PROGRAM Pneumatics_Template_Shutter
VAR
    bExtendedLight AT %Q*: BOOL; //Power output for Open position + LED
    bRetractedLight AT %Q*: BOOL; //Power output for Close position + LED
    bMovingLight AT %Q*: BOOL; //Power output for cylinder Moving LED
    bNoPermitLight AT %Q*: BOOL; //Power output for No permit LED
    bErrorLight AT %Q*: BOOL; //Power output for Error LED
END_VAR

//Assign LED to the permit status
bNoPermitLight := NOT gvl.astPneumaticAxes[main.hmiPneumaticAxisSelection].stPneumaticAxisInputs.bPSSPermit;

//Assign LED to the error status
bErrorLight := gvl.astPneumaticAxes[main.hmiPneumaticAxisSelection].stPneumaticAxisStatus.bError;

//Assign LEDs to the end switches statuses
bExtendedLight := gvl.astPneumaticAxes[main.hmiPneumaticAxisSelection].stPneumaticAxisStatus.bExtended;
bRetractedLight := gvl.astPneumaticAxes[main.hmiPneumaticAxisSelection].stPneumaticAxisStatus.bRetracted;

//Checking the condition for the Moving LED
IF gvl.astPneumaticAxes[main.hmiPneumaticAxisSelection].stPneumaticAxisStatus.bRetracting OR gvl.astPneumaticAxes[main.hmiPneumaticAxisSelection].stPneumaticAxisStatus.bExtending THEN
        bMovingLight := TRUE;
    ELSE
        bMovingLight := FALSE;
    END_IF

END_PROGRAM

(* stored: Version 1.1.0.1, ProductVersion 3.1.4024.11
   POU Pneumatics_Template_Shutter: Id {f0d41dcb-32b4-49cb-acfd-0a4b7f2819f3}, SpecialFunc None *)
